{attribute 'no_explicit_call'} 
FUNCTION_BLOCK PUBLIC FB_Observer IMPLEMENTS I_Observer
VAR
	pList: 			POINTER TO I_Component;
	nLength:		DINT;
	aList:			POINTER TO POINTER TO ARRAY [0..100] OF I_Component:=ADR(pList);
END_VAR

METHOD FB_exit : BOOL
VAR_INPUT
	bInCopyCode : BOOL; // if TRUE, the exit method is called for exiting an instance that is copied afterwards (online change).
END_VAR
M_Clear();
END_METHOD

METHOD M_Attach : BOOL
VAR_INPUT
	Object: 	I_Component;
END_VAR
VAR
	pOldList: 	POINTER TO I_Component;
END_VAR
IF Object <> 0 THEN
	// First Item
	IF pList = 0 THEN
		nLength:= nLength + 1;
		pList:= __NEW(POINTER TO I_Component,DINT_TO_UDINT(nLength));
	ELSE
		// Item already in List
		IF M_Find(Object) = -1 THEN
			// backup 
			pOldList:= pList;
			// new Length
			nLength:= nLength + 1;
			// new pointer
			pList:= __NEW(POINTER TO I_Component,DINT_TO_UDINT(nLength));
			// restore
			Memcpy(pList,pOldList, SIZEOF(POINTER TO I_Component)*DINT_TO_UDINT(nLength -1));
			// delete old
			__DELETE(pOldList);
		ELSE
			M_Attach:= FALSE;	
			RETURN;
		END_IF
	END_IF
	IF pList = 0 THEN
		RETURN;
	END_IF
	// add new Object
	pList[nLength-1]:= Object;
	M_Attach:= TRUE;
ELSE
	M_Attach:= FALSE;	
END_IF
END_METHOD

METHOD M_Clear
IF pList <> 0 THEN
	nLength:= 0;
	__DELETE(pList);
END_IF
END_METHOD

METHOD M_Detach : BOOL
VAR_INPUT
	Object: 	I_Component;
END_VAR
VAR
	pOldList:			POINTER TO I_Component;
	nPosition: 			DINT;
END_VAR
IF Object <> 0 THEN
	// First Item
	IF nLength >= 0 THEN
		// Item already in List
		nPosition:= M_Find(Object);
		IF nPosition <> -1 THEN
			// backup 
			pOldList:= pList;
			// new Length
			nLength:= nLength -1;
			// new pointer
			pList:= __NEW(POINTER TO I_Component,DINT_TO_UDINT(nLength));
			// restore lower part
			Memcpy(pList,pOldList, SIZEOF(POINTER TO I_Component) * DINT_TO_UDINT(nPosition));
			//pList[nPosition]:= iObject;
			Memcpy(pList + (SIZEOF(POINTER TO I_Component)*nPosition),pOldList + (SIZEOF(POINTER TO I_Component)*(nPosition + 1)), SIZEOF(POINTER TO I_Component) * DINT_TO_UDINT(nLength - nPosition));
			// delete old
			__DELETE(pOldList);
		ELSE
			M_Detach:= FALSE;	
			RETURN;
		END_IF
	ELSE
		M_Detach:= FALSE;	
		RETURN;
	END_IF
	M_Detach:= TRUE;
ELSE
	M_Detach:= FALSE;	
END_IF
END_METHOD

METHOD M_Find : DINT
VAR_INPUT
	Object: 	I_Component;
END_VAR
VAR
	nIndex: 	UINT;
END_VAR
// Object already in List
M_Find := -1;
WHILE nIndex < nLength DO
    IF (pList[nIndex] = Object) THEN
        M_Find := nIndex;
        RETURN;
    END_IF
	nIndex := nIndex + 1;
END_WHILE
END_METHOD

METHOD M_Index : I_Component
VAR_INPUT
	Index: 	DINT;
END_VAR
IF Index <= nLength THEN
	M_Index:= pList[Index];
END_IF
END_METHOD

METHOD M_Notify : BOOL
VAR_INPUT
	eRequest:		E_Request;
END_VAR

VAR
	nIndex: 	INT;
END_VAR
WHILE nIndex < nLength DO
	pList[nIndex].M_Request(eRequest);
	nIndex:= nIndex + 1; 
END_WHILE
END_METHOD

PROPERTY P_Length : DINT
GET
P_Length:= nLength;
END_GET
END_PROPERTY

END_FUNCTION_BLOCK

(* stored: Version 1.1.0.1
   POU FB_Observer: Id {52aee6c6-b98c-4cb9-9b9b-2f523841c4cc}, SpecialFunc None
   Method FB_exit: Id {8920c8e0-5709-4e5e-a21f-0871704cdcd1}
   Method M_Attach: Id {a96df4cc-8cea-4396-beb7-115ce888674b}
   Method M_Clear: Id {307f5dd9-2a35-4b04-93bb-a7de0406e653}
   Method M_Detach: Id {6e982e5c-8b12-4999-bbf2-06e2eebe2934}
   Method M_Find: Id {315829c2-37f1-487f-acb0-fff200e1a3d8}
   Method M_Index: Id {6e332950-284b-4ced-bcaa-31bfc1d4668b}
   Method M_Notify: Id {3d3fb67b-dd6a-440b-9c1c-e8b43c7588bf}
   Property P_Length: Id {8da11863-b503-4855-a3f1-c1f64dac07a1}
   Get Get: Id {81573980-0484-490c-84fc-be91d0b14826} *)
